{attribute 'qualified_only'}
VAR_GLOBAL
	arrId	AT %I*:	ARRAY[0..255] OF UINT;
END_VAR

(* stored: Version 1.1.0.1, ProductVersion 3.1.4024.6
   GVL GVL_IO: Id {24b51e13-7c95-495e-a450-4e3643e19705} *)
